(* IEC 61131-3 sources: CodesysTest/export/SX_1195.dev/Plc Logic/Application/PRJ Specific/Motion/Motors/Applied Motion/Applied Motion TSM34IP-3DG/FB_BaseAppliedMotionMotorEIP.pou/ScaledProfileTargetPostion.prop, 1 file *)

(* ---- Get.pm.st ---- *)
(*#-#-#-#-#-#-#-#-#-#---Declaration---#-#-#-#-#-#-#-#-#-#-#-#-#*)

VAR
END_VAR
(*#-#-#-#-#-#-#-#-#-#---Implementation---#-#-#-#-#-#-#-#-#-#-#-#-#*)

ScaledProfileTargetPostion := targetPosDist * TO_REAL(stepsPerInch);
IF reversePolarity THEN
	ScaledProfileTargetPostion := ScaledProfileTargetPostion * -1;
END_IF
